Yaskawa INFORM job: R1_W35-36-A1(90,180)KM-OK.JBI

/JOB
//NAME R1_W35-36-A1(90,180)KM-OK
///FOLDERNAME KRIS-SCIANA
//POS
///NPOS 72,72,0,4,0,0
///TOOL 0
///POSTYPE PULSE
///PULSE
C00000=105585,-55022,-75652,10862,69152,39815
C00001=105585,-55022,-75652,10862,69152,39815
C00002=25297,-64730,-92267,55168,72656,-59021
C00003=33428,-24381,-57031,51925,58941,-79758
C00004=40351,-25600,-48168,51274,51402,-80679
C00005=41423,-24438,-46515,50909,50557,-80585
C00006=42396,-23179,-45620,50269,50100,-80278
C00007=41423,-24438,-46515,50909,50557,-80585
C00008=52197,-27156,-57835,19815,52622,-73041
C00009=52201,-27467,-57246,19946,52129,-73139
C00010=52197,-27156,-57835,19815,52622,-73041
C00011=51548,-28474,-59924,20162,53342,-73162
C00012=49863,-31663,-65047,21063,55152,-73465
C00013=115393,-122942,-108395,-21741,33563,-54940
C00014=115738,-113039,-102237,-21412,34866,-55128
C00015=115865,-109374,-99803,-21347,35259,-55169
C00016=115984,-105750,-98521,-20934,36294,-55402
C00017=115865,-109374,-99803,-21347,35259,-55169
C00018=100189,-107821,-99394,13346,35679,-69154
C00019=100201,-107595,-98316,13511,35145,-69245
C00020=100189,-107821,-99394,13346,35679,-69154
C00021=99280,-111033,-101668,14411,35591,-69703
C00022=96833,-119539,-107384,17358,35244,-71233
C00023=105118,-107156,-116180,-7812,55751,-63740
C00024=88402,-92633,-103842,3937,55232,-70237
C00025=85657,-85306,-98934,5813,56133,-71264
C00026=85657,-85601,-98129,5854,55490,-71299
C00027=85657,-85306,-98934,5813,56133,-71264
C00028=88898,-98879,-97009,8739,38201,-70578
C00029=89964,-94121,-94598,7471,39048,-69926
C00030=90400,-92130,-93799,6947,39535,-69656
C00031=89774,-94980,-95242,7673,39023,-70029
C00032=72922,-111625,-112899,22845,44407,-77640
C00033=76129,-93837,-107755,-10075,52469,-61366
C00034=80813,-77974,-91117,-30690,51731,-50959
C00035=85919,-63418,-71861,-50871,54293,-42403
C00036=85689,-63243,-70894,-51038,53840,-42243
C00037=84470,-62094,-70296,-50310,53321,-42659
C00038=85689,-63243,-70894,-51038,53840,-42243
C00039=92588,-72277,-84322,-52450,59930,-42067
C00040=73945,-93495,-114912,-15532,68902,-60225
C00041=58434,-53005,-100968,5225,92482,-77281
C00042=58848,-52643,-94168,5049,88476,-77324
C00043=82964,-48312,-91591,-4565,89053,-70386
C00044=82850,-44336,-94003,-4534,92565,-70546
C00045=69976,-54144,-97914,-9670,89664,-77094
C00046=71132,-53816,-94045,-10127,87600,-76594
C00047=45687,-49511,-91635,272,86979,-83967
C00048=45786,-46119,-93680,232,89981,-83932
C00049=37246,-30334,-87191,12662,99095,-84829
C00050=20453,-12601,-69080,36945,106911,-87667
C00051=18131,3710,-49188,45242,115448,-83422
C00052=23953,6560,-47103,43203,113198,-82423
C00053=27421,-9079,-69038,35213,106037,-85552
C00054=66885,-25870,-83180,7915,99205,-66136
C00055=68322,-30750,-82029,7327,95908,-65941
C00056=89648,-22173,-76277,-390,96021,-60015
C00057=85856,-24196,-83471,1007,99418,-61035
C00058=54513,-23053,-67930,19868,75683,-58524
C00059=56472,-21312,-63598,18974,73603,-58237
C00060=57193,-19604,-61763,18606,73218,-58067
C00061=56423,-22124,-62953,19075,72841,-58376
C00062=57225,-19765,-62562,18556,73600,-57993
C00063=58084,-17666,-61706,18118,76143,-57272
C00064=57991,-17929,-61778,18175,76074,-57312
C00065=57215,-19459,-61291,18615,73007,-58089
C00066=56490,-21147,-63697,18951,73738,-58209
C00067=54532,-22872,-68023,19845,75820,-58495
C00068=48154,-122420,-119423,19643,55864,-58497
C00069=113071,-122345,-116911,19991,54442,-58776
C00070=113071,-122345,-116911,19991,54442,-58776
C00071=-3488,-122345,-116911,19991,54442,-58776
BC00000=6655,833354,935576
BC00001=6655,1280278,935576
BC00002=29793,1210760,1039028
BC00003=36322,1191142,1068222
BC00004=36322,1191142,1068222
BC00005=36322,1191142,1068222
BC00006=36322,1191142,1068222
BC00007=36322,1191142,1068222
BC00008=36322,1191142,1068222
BC00009=36322,1191142,1068222
BC00010=36322,1191142,1068222
BC00011=36322,1191142,1068222
BC00012=36322,1191142,1068222
BC00013=146609,1191142,1068222
BC00014=146609,1191142,1068222
BC00015=146609,1191142,1068222
BC00016=146609,1191142,1068222
BC00017=146609,1191142,1068222
BC00018=146609,1191142,1068222
BC00019=146609,1191142,1068222
BC00020=146609,1191142,1068222
BC00021=146609,1191142,1068222
BC00022=146609,1191142,1068222
BC00023=146609,1191142,1068222
BC00024=146609,1191142,1068222
BC00025=146609,1191142,1068222
BC00026=146609,1191142,1068222
BC00027=146609,1191142,1068222
BC00028=146609,1191142,1068222
BC00029=146609,1191142,1068222
BC00030=146609,1191142,1068222
BC00031=146609,1191142,1068222
BC00032=146609,1191142,1068222
BC00033=146609,1191142,1068222
BC00034=146609,1191142,1068222
BC00035=146609,1191142,1068222
BC00036=146609,1191142,1068222
BC00037=146609,1191142,1068222
BC00038=146609,1191142,1068222
BC00039=146609,1191142,1068222
BC00040=145056,1191142,1068222
BC00041=143373,1191142,1068222
BC00042=143373,1191142,1068222
BC00043=143373,1191142,1068222
BC00044=143373,1191142,1068222
BC00045=143373,1191142,1068222
BC00046=143373,1191142,1068222
BC00047=143373,1191142,1068222
BC00048=143373,1191142,1068222
BC00049=143373,1191142,1068222
BC00050=143373,1191142,1068222
BC00051=143373,1191142,1068222
BC00052=143373,1191142,1068222
BC00053=143373,1191142,1068222
BC00054=127887,1191142,1068222
BC00055=127887,1191142,1068222
BC00056=127887,1191142,1068222
BC00057=127887,1191142,1068222
BC00058=70873,1191142,1068222
BC00059=70144,1191142,1068222
BC00060=69852,1191142,1068222
BC00061=69852,1191142,1068222
BC00062=69852,1191142,1068222
BC00063=58916,1191142,1068222
BC00064=55589,1191142,1068222
BC00065=20480,1191142,1068222
BC00066=20771,1191142,1068222
BC00067=21500,1191142,1068222
BC00068=21500,1191142,1068221
BC00069=21500,1384690,1084351
BC00070=21500,863244,1084351
BC00071=22430,863244,1084351
///POSTYPE BASE
///RECTAN
///RCONF 0,0,0,0,0,0,0,0,0,0,0,0,0,0,0,0,0,0,0,0,0,0,0,0
P00006=0.222,-3.123,-1.508,0.0000,0.0000,0.0000
P00021=-0.225,-6.128,-0.405,0.0000,0.0000,0.0000
P00022=0.222,-3.123,-1.508,0.0000,0.0000,0.0000
P00030=5.926,-4.294,-1.390,0.0000,0.0000,0.0000
//INST
///DATE 2024/07/25 09:59
///ATTR SC,RW
///GROUP1 RB1,BS1
NOP
'r1_W35-36-A1(90,180)
'Path S1030 (for W465)
SFTOF
MOVJ C00000 BC00000 VJ=50.00
MOVJ C00001 BC00001 VJ=50.00
MOVJ C00002 BC00002 VJ=50.00
MOVJ C00003 BC00003 VJ=40.00
MOVJ C00004 BC00004 VJ=20.00
MOVL C00005 BC00005 V=60.0
REFP 3 C00006 BC00006
CALL JOB:SEARCH-R1
SET P021 P006
SFTON P021
MOVL C00007 BC00007 V=60.0
MOVL C00008 BC00008 V=60.0
REFP 3 C00009 BC00009
CALL JOB:SEARCH-R1
SET P021 P006
SFTON P021
MOVL C00010 BC00010 V=60.0
MOVL C00011 BC00011 V=166.7
MOVL C00012 BC00012 V=166.7
'Path S1031 (for W465)
SFTOF
MOVL C00013 BC00013 V=166.7
MOVL C00014 BC00014 V=166.7
MOVL C00015 BC00015 V=60.0
REFP 3 C00016 BC00016
CALL JOB:SEARCH-R1
SET P022 P006
SFTON P022
MOVL C00017 BC00017 V=60.0
MOVL C00018 BC00018 V=60.0
REFP 3 C00019 BC00019
CALL JOB:SEARCH-R1
SET P022 P006
SFTON P022
MOVL C00020 BC00020 V=60.0
MOVL C00021 BC00021 V=166.7
MOVL C00022 BC00022 V=166.7
'Path VIA1148
SFTOF
MOVJ C00023 BC00023 VJ=20.00
MOVJ C00024 BC00024 VJ=10.00
MOVL C00025 BC00025 V=83.3
REFP 3 C00026 BC00026
CALL JOB:SEARCH-R1
SET P030 P006
SFTON P030
MOVL C00027 BC00027 V=83.3
MOVJ C00028 BC00028 VJ=10.00
MOVL C00029 BC00029 V=66.7
REFP 3 C00030 BC00030
CALL JOB:SEARCH-R1
SET P030 P006
SFTON P030
MOVL C00031 BC00031 V=83.3
MOVJ C00032 BC00032 VJ=50.00
MOVJ C00033 BC00033 VJ=50.00
MOVJ C00034 BC00034 VJ=50.00
MOVJ C00035 BC00035 VJ=50.00
MOVL C00036 BC00036 V=66.7
REFP 3 C00037 BC00037
CALL JOB:SEARCH-R1
SET P030 P006
SFTON P030
MOVL C00038 BC00038 V=83.3
MOVJ C00039 BC00039 VJ=50.00
MOVJ C00040 BC00040 VJ=50.00
SFTOF
MOVJ C00041 BC00041 VJ=10.00
SFTON P030
MACRO1 MJ#(0) ARGF7
MOVJ C00042 BC00042 VJ=10.00
ARCON
MOVL C00043 BC00043 V=11.7
ARCOF
MOVJ C00044 BC00044 VJ=10.00
MOVJ C00045 BC00045 VJ=60.00
MOVJ C00046 BC00046 VJ=10.00
ARCON
MOVL C00047 BC00047 V=11.7
ARCOF
MOVJ C00048 BC00048 VJ=10.00
MOVJ C00049 BC00049 VJ=10.00
MOVJ C00050 BC00050 VJ=10.00
MACRO1 MJ#(0) ARGF6
MOVJ C00051 BC00051 VJ=10.00
MOVL C00052 BC00052 V=11.7
ARCOF
MOVJ C00053 BC00053 VJ=10.00
MOVJ C00054 BC00054 VJ=20.00
MACRO1 MJ#(0) ARGF7
MOVJ C00055 BC00055 VJ=10.00
ARCON
MOVL C00056 BC00056 V=11.7
ARCOF
MOVJ C00057 BC00057 VJ=10.00
'Path W1032
SFTOF
SFTON P022
MOVJ C00058 BC00058 VJ=20.00
MOVJ C00059 BC00059 VJ=20.00
MOVL C00060 BC00060 V=166.7 PL=0
REFP 1 C00061 BC00061
REFP 2 C00062 BC00062
MACRO1 MJ#(0) ARGF7
ARCON
MOVL C00063 BC00063 V=7.5
SFTON P021
MOVL C00064 BC00064 V=7.5
MOVL C00065 BC00065 V=7.5
ARCOF
MOVL C00066 BC00066 V=166.7
MOVL C00067 BC00067 V=250.0
SFTOF
MOVJ C00068 BC00068 VJ=80.00
COMM MOVJ C00069 BC00069 VJ=100.00
COMM MOVJ C00070 BC00070 VJ=100.00
COMM MOVJ C00071 BC00071 VJ=100.00
END
